// Phase 0 - E_WS_State
// Rev 1.0 - January 8, 2024

TYPE E_WS_State :
(
	eWSIdle			 													:= 0,
	eWSReadCoils,
	eWSReadInputStatus,
	eWSReadRegs,
	eWSReadInputRegs,
	eWSWriteSingleCoil,
	eWSWriteSingleReg,
	eWSWriteMultipleCoils,
	eWSWriteRegs
);
END_TYPE

(* stored: Version 1.1.0.1, ProductVersion 3.1.4024.12
   DUT E_WS_State: Id {091a3451-a681-4903-9548-847951b61c62} *)
